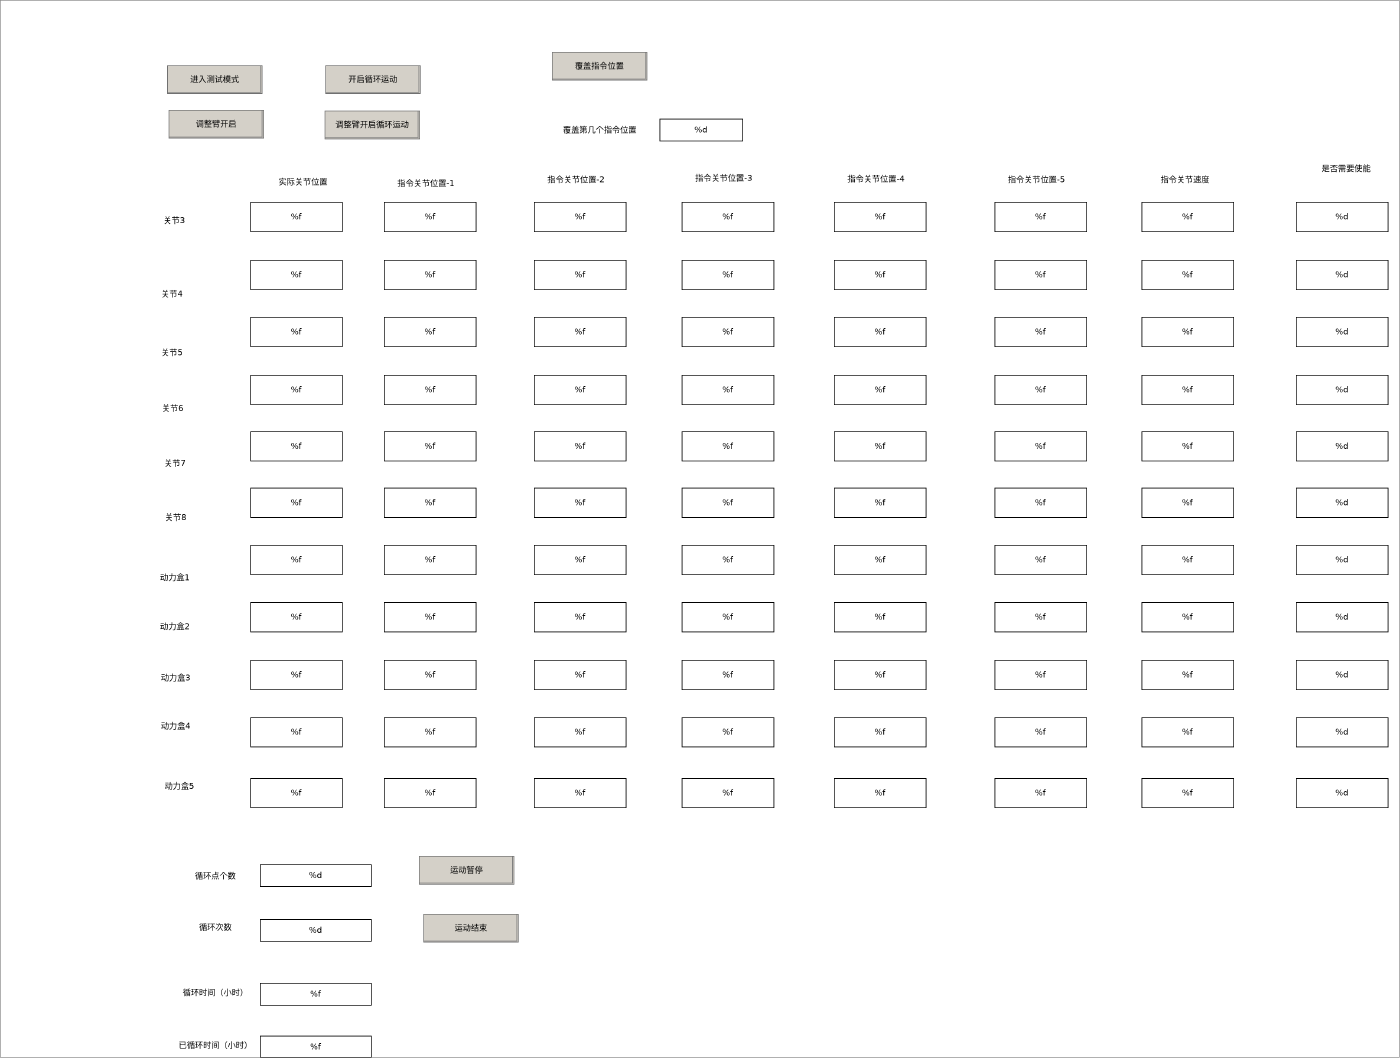
VISUALIZATION cycle_a1  // 1885x1425
    Button (225,88 128x38), "进入测试模式", colour toggle: g_cycleTest.m_enterCycleTestMode[1]
        toggle g_cycleTest.m_enterCycleTestMode[1]
    Button (438,88 128x38), "开启循环运动", colour toggle: g_cycleTest.m_startMotion[1]
        toggle g_cycleTest.m_startMotion[1]
    Label (215,1165 150x30), "循环点个数"
    Rectangle (350,1164 150x30), "%d", text variable: g_cycleTest.m_pointSum[1]
        OnMouseClick: write the text variable via Default
    Rectangle (350,1238 150x30), "%d", text variable: g_cycleTest.m_curCycleNum[1]
    Label (215,1234 150x30), "循环次数"
    Button (564,1153 128x38), "运动暂停", colour toggle: g_cycleTest.m_pause[1]
        toggle g_cycleTest.m_pause[1]
    Button (570,1231 128x38), "运动结束", colour toggle: g_cycleTest.m_finish[1]
        tap g_cycleTest.m_finish[1]
    Label (501,233 145x28), "指令关节位置-1"
    Label (333,230 150x30), "实际关节位置"
    Rectangle (337,505 124x40), "%f", text variable: g_cycleTest.m_actJntPos[1][1]
    Label (162,283 145x28), "关节3"
    Label (159,382 145x28), "关节4"
    Label (159,461 145x28), "关节5"
    Label (160,536 145x28), "关节6"
    Label (163,610 145x28), "关节7"
    Label (164,683 145x28), "关节8"
    Label (163,764 145x28), "动力盒1"
    Label (163,830 145x28), "动力盒2"
    Label (169,1045 145x28), "动力盒5"
    Label (164,899 145x28), "动力盒3"
    Label (164,964 145x28), "动力盒4"
    Rectangle (337,581 124x40), "%f", text variable: g_cycleTest.m_actJntPos[1][2]
    Rectangle (337,657 124x40), "%f", text variable: g_cycleTest.m_actJntPos[1][3]
    Rectangle (337,734 124x40), "%f", text variable: g_cycleTest.m_actJntPos[1][4]
    Rectangle (337,811 124x40), "%f", text variable: g_cycleTest.m_actJntPos[1][5]
    Rectangle (337,889 124x40), "%f", text variable: g_cycleTest.m_actJntPos[1][6]
    Rectangle (337,966 124x40), "%f", text variable: g_cycleTest.m_actJntPos[1][7]
    Rectangle (337,1048 124x40), "%f", text variable: g_cycleTest.m_actJntPos[1][8]
    Rectangle (337,272 124x40), "%f", text variable: g_cycleTest.m_actJntPosSetup[1][3]
    Rectangle (337,350 124x40), "%f", text variable: g_cycleTest.m_actJntPosSetup[1][4]
    Rectangle (337,427 124x40), "%f", text variable: g_cycleTest.m_actJntPosSetup[1][5]
    Rectangle (517,272 124x40), "%f", text variable: g_cycleTest.m_targetJntPosSetup[1,1][3]
        OnMouseClick: write the text variable via Default
    Rectangle (517,350 124x40), "%f", text variable: g_cycleTest.m_targetJntPosSetup[1,1][4]
        OnMouseClick: write the text variable via Default
    Rectangle (517,427 124x40), "%f", text variable: g_cycleTest.m_targetJntPosSetup[1,1][5]
        OnMouseClick: write the text variable via Default
    Rectangle (517,505 124x40), "%f", text variable: g_cycleTest.m_targetJntPos[1,1][1]
        OnMouseClick: write the text variable via Default
    Rectangle (517,581 124x40), "%f", text variable: g_cycleTest.m_targetJntPos[1,1][2]
        OnMouseClick: write the text variable via Default
    Rectangle (517,657 124x40), "%f", text variable: g_cycleTest.m_targetJntPos[1,1][3]
        OnMouseClick: write the text variable via Default
    Rectangle (517,734 124x40), "%f", text variable: g_cycleTest.m_targetJntPos[1,1][4]
        OnMouseClick: write the text variable via Default
    Rectangle (517,811 124x40), "%f", text variable: g_cycleTest.m_targetJntPos[1,1][5]
        OnMouseClick: write the text variable via Default
    Rectangle (517,889 124x40), "%f", text variable: g_cycleTest.m_targetJntPos[1,1][6]
        OnMouseClick: write the text variable via Default
    Rectangle (517,966 124x40), "%f", text variable: g_cycleTest.m_targetJntPos[1,1][7]
        OnMouseClick: write the text variable via Default
    Rectangle (517,1048 124x40), "%f", text variable: g_cycleTest.m_targetJntPos[1,1][8]
        OnMouseClick: write the text variable via Default
    Label (703,228 145x28), "指令关节位置-2"
    Rectangle (719,272 124x40), "%f", text variable: g_cycleTest.m_targetJntPosSetup[1,2][3]
        OnMouseClick: write the text variable via Default
    Rectangle (719,350 124x40), "%f", text variable: g_cycleTest.m_targetJntPosSetup[1,2][4]
        OnMouseClick: write the text variable via Default
    Rectangle (719,427 124x40), "%f", text variable: g_cycleTest.m_targetJntPosSetup[1,2][5]
        OnMouseClick: write the text variable via Default
    Rectangle (719,505 124x40), "%f", text variable: g_cycleTest.m_targetJntPos[1,2][1]
        OnMouseClick: write the text variable via Default
    Rectangle (719,581 124x40), "%f", text variable: g_cycleTest.m_targetJntPos[1,2][2]
        OnMouseClick: write the text variable via Default
    Rectangle (719,657 124x40), "%f", text variable: g_cycleTest.m_targetJntPos[1,2][3]
        OnMouseClick: write the text variable via Default
    Rectangle (719,734 124x40), "%f", text variable: g_cycleTest.m_targetJntPos[1,2][4]
        OnMouseClick: write the text variable via Default
    Rectangle (719,811 124x40), "%f", text variable: g_cycleTest.m_targetJntPos[1,2][5]
        OnMouseClick: write the text variable via Default
    Rectangle (719,889 124x40), "%f", text variable: g_cycleTest.m_targetJntPos[1,2][6]
        OnMouseClick: write the text variable via Default
    Rectangle (719,966 124x40), "%f", text variable: g_cycleTest.m_targetJntPos[1,2][7]
        OnMouseClick: write the text variable via Default
    Rectangle (719,1048 124x40), "%f", text variable: g_cycleTest.m_targetJntPos[1,2][8]
        OnMouseClick: write the text variable via Default
    Label (902,226 145x28), "指令关节位置-3"
    Rectangle (918,272 124x40), "%f", text variable: g_cycleTest.m_targetJntPosSetup[1,3][3]
        OnMouseClick: write the text variable via Default
    Rectangle (918,350 124x40), "%f", text variable: g_cycleTest.m_targetJntPosSetup[1,3][4]
        OnMouseClick: write the text variable via Default
    Rectangle (918,427 124x40), "%f", text variable: g_cycleTest.m_targetJntPosSetup[1,3][5]
        OnMouseClick: write the text variable via Default
    Rectangle (918,505 124x40), "%f", text variable: g_cycleTest.m_targetJntPos[1,3][1]
        OnMouseClick: write the text variable via Default
    Rectangle (918,581 124x40), "%f", text variable: g_cycleTest.m_targetJntPos[1,3][2]
        OnMouseClick: write the text variable via Default
    Rectangle (918,657 124x40), "%f", text variable: g_cycleTest.m_targetJntPos[1,3][3]
        OnMouseClick: write the text variable via Default
    Rectangle (918,734 124x40), "%f", text variable: g_cycleTest.m_targetJntPos[1,3][4]
        OnMouseClick: write the text variable via Default
    Rectangle (918,811 124x40), "%f", text variable: g_cycleTest.m_targetJntPos[1,3][5]
        OnMouseClick: write the text variable via Default
    Rectangle (918,889 124x40), "%f", text variable: g_cycleTest.m_targetJntPos[1,3][6]
        OnMouseClick: write the text variable via Default
    Rectangle (918,966 124x40), "%f", text variable: g_cycleTest.m_targetJntPos[1,3][7]
        OnMouseClick: write the text variable via Default
    Rectangle (918,1048 124x40), "%f", text variable: g_cycleTest.m_targetJntPos[1,3][8]
        OnMouseClick: write the text variable via Default
    Label (1107,227 145x28), "指令关节位置-4"
    Rectangle (1123,272 124x40), "%f", text variable: g_cycleTest.m_targetJntPosSetup[1,4][3]
        OnMouseClick: write the text variable via Default
    Rectangle (1123,350 124x40), "%f", text variable: g_cycleTest.m_targetJntPosSetup[1,4][4]
        OnMouseClick: write the text variable via Default
    Rectangle (1123,427 124x40), "%f", text variable: g_cycleTest.m_targetJntPosSetup[1,4][5]
        OnMouseClick: write the text variable via Default
    Rectangle (1123,505 124x40), "%f", text variable: g_cycleTest.m_targetJntPos[1,4][1]
        OnMouseClick: write the text variable via Default
    Rectangle (1123,581 124x40), "%f", text variable: g_cycleTest.m_targetJntPos[1,4][2]
        OnMouseClick: write the text variable via Default
    Rectangle (1123,657 124x40), "%f", text variable: g_cycleTest.m_targetJntPos[1,4][3]
        OnMouseClick: write the text variable via Default
    Rectangle (1123,734 124x40), "%f", text variable: g_cycleTest.m_targetJntPos[1,4][4]
        OnMouseClick: write the text variable via Default
    Rectangle (1123,811 124x40), "%f", text variable: g_cycleTest.m_targetJntPos[1,4][5]
        OnMouseClick: write the text variable via Default
    Rectangle (1123,889 124x40), "%f", text variable: g_cycleTest.m_targetJntPos[1,4][6]
        OnMouseClick: write the text variable via Default
    Rectangle (1123,966 124x40), "%f", text variable: g_cycleTest.m_targetJntPos[1,4][7]
        OnMouseClick: write the text variable via Default
    Rectangle (1123,1048 124x40), "%f", text variable: g_cycleTest.m_targetJntPos[1,4][8]
        OnMouseClick: write the text variable via Default
    Label (1323,228 145x28), "指令关节位置-5"
    Rectangle (1339,272 124x40), "%f", text variable: g_cycleTest.m_targetJntPosSetup[1,5][3]
        OnMouseClick: write the text variable via Default
    Rectangle (1339,350 124x40), "%f", text variable: g_cycleTest.m_targetJntPosSetup[1,5][4]
        OnMouseClick: write the text variable via Default
    Rectangle (1339,427 124x40), "%f", text variable: g_cycleTest.m_targetJntPosSetup[1,5][5]
        OnMouseClick: write the text variable via Default
    Rectangle (1339,505 124x40), "%f", text variable: g_cycleTest.m_targetJntPos[1,5][1]
        OnMouseClick: write the text variable via Default
    Rectangle (1339,581 124x40), "%f", text variable: g_cycleTest.m_targetJntPos[1,5][2]
        OnMouseClick: write the text variable via Default
    Rectangle (1339,657 124x40), "%f", text variable: g_cycleTest.m_targetJntPos[1,5][3]
        OnMouseClick: write the text variable via Default
    Rectangle (1339,734 124x40), "%f", text variable: g_cycleTest.m_targetJntPos[1,5][4]
        OnMouseClick: write the text variable via Default
    Rectangle (1339,811 124x40), "%f", text variable: g_cycleTest.m_targetJntPos[1,5][5]
        OnMouseClick: write the text variable via Default
    Rectangle (1339,889 124x40), "%f", text variable: g_cycleTest.m_targetJntPos[1,5][6]
        OnMouseClick: write the text variable via Default
    Rectangle (1339,966 124x40), "%f", text variable: g_cycleTest.m_targetJntPos[1,5][7]
        OnMouseClick: write the text variable via Default
    Rectangle (1339,1048 124x40), "%f", text variable: g_cycleTest.m_targetJntPos[1,5][8]
        OnMouseClick: write the text variable via Default
    Button (227,148 128x38), "调整臂开启", colour toggle: g_cycleTest.m_enterCycleTestModeSetup[1]
        toggle g_cycleTest.m_enterCycleTestModeSetup[1]
    Button (437,149 128x38), "调整臂开启循环运动", colour toggle: g_cycleTest.m_startMotionSetup[1]
        toggle g_cycleTest.m_startMotionSetup[1]
    Button (743,70 128x38), "覆盖指令位置", colour toggle: g_cycleTest.m_coverCmdPos[1]
        tap g_cycleTest.m_coverCmdPos[1]
    Rectangle (888,160 112x30), "%d", text variable: g_cycleTest.m_pntIdForCoverCmd[1]
        OnMouseClick: write the text variable via Default
    Label (735,161 145x28), "覆盖第几个指令位置"
    Label (1523,228 145x28), "指令关节速度"
    Rectangle (1537,272 124x40), "%f", text variable: g_cycleTest.m_targetJntVelSetup[1][3]
        OnMouseClick: write the text variable via Default
    Rectangle (1537,350 124x40), "%f", text variable: g_cycleTest.m_targetJntVelSetup[1][4]
        OnMouseClick: write the text variable via Default
    Rectangle (1537,427 124x40), "%f", text variable: g_cycleTest.m_targetJntVelSetup[1][5]
        OnMouseClick: write the text variable via Default
    Rectangle (1537,505 124x40), "%f", text variable: g_cycleTest.m_targetJntVelN8[1][1]
        OnMouseClick: write the text variable via Default
    Rectangle (1537,581 124x40), "%f", text variable: g_cycleTest.m_targetJntVelN8[1][2]
        OnMouseClick: write the text variable via Default
    Rectangle (1537,657 124x40), "%f", text variable: g_cycleTest.m_targetJntVelN8[1][3]
        OnMouseClick: write the text variable via Default
    Rectangle (1537,734 124x40), "%f", text variable: g_cycleTest.m_targetJntVelN8[1][4]
        OnMouseClick: write the text variable via Default
    Rectangle (1537,811 124x40), "%f", text variable: g_cycleTest.m_targetJntVelN8[1][5]
        OnMouseClick: write the text variable via Default
    Rectangle (1537,889 124x40), "%f", text variable: g_cycleTest.m_targetJntVelN8[1][6]
        OnMouseClick: write the text variable via Default
    Rectangle (1537,966 124x40), "%f", text variable: g_cycleTest.m_targetJntVelN8[1][7]
        OnMouseClick: write the text variable via Default
    Rectangle (1537,1048 124x40), "%f", text variable: g_cycleTest.m_targetJntVelN8[1][8]
        OnMouseClick: write the text variable via Default
    Rectangle (350,1324 150x30), "%f", text variable: g_cycleTest.m_tgtCycleTime[1]
        OnMouseClick: write the text variable via Default
    Label (215,1322 150x30), "循环时间（小时）"
    Rectangle (350,1395 150x30), "%f", text variable: g_cycleTest.m_curCycleTime[1]
        OnMouseClick: write the text variable via Default
    Label (215,1393 150x30), "已循环时间（小时）"
    Label (1740,212 145x30), "是否需要使能"
    Rectangle (1745,272 124x40), "%d", text variable: g_cycleTest.m_jntEnableSetup[1][3]
        OnMouseClick: write the text variable via Default
    Rectangle (1745,350 124x40), "%d", text variable: g_cycleTest.m_jntEnableSetup[1][4]
        OnMouseClick: write the text variable via Default
    Rectangle (1745,427 124x40), "%d", text variable: g_cycleTest.m_jntEnableSetup[1][5]
        OnMouseClick: write the text variable via Default
    Rectangle (1745,505 124x40), "%d", text variable: g_cycleTest.m_jntEnable[1][1]
        OnMouseClick: write the text variable via Default
    Rectangle (1745,581 124x40), "%d", text variable: g_cycleTest.m_jntEnable[1][2]
        OnMouseClick: write the text variable via Default
    Rectangle (1745,657 124x40), "%d", text variable: g_cycleTest.m_jntEnable[1][3]
        OnMouseClick: write the text variable via Default
    Rectangle (1745,734 124x40), "%d", text variable: g_cycleTest.m_jntEnable[1][4]
        OnMouseClick: write the text variable via Default
    Rectangle (1745,811 124x40), "%d", text variable: g_cycleTest.m_jntEnable[1][5]
        OnMouseClick: write the text variable via Default
    Rectangle (1745,889 124x40), "%d", text variable: g_cycleTest.m_jntEnable[1][6]
        OnMouseClick: write the text variable via Default
    Rectangle (1745,966 124x40), "%d", text variable: g_cycleTest.m_jntEnable[1][7]
        OnMouseClick: write the text variable via Default
    Rectangle (1745,1048 124x40), "%d", text variable: g_cycleTest.m_jntEnable[1][8]
        OnMouseClick: write the text variable via Default
END_VISUALIZATION

(* stored: Version 1.1.0.1, ProductVersion 3.1.4024.11
   Visu cycle_a1: Id {9697ab1e-d88f-406f-a5ae-e8f833fc7269} *)
